// TIA Portal V16 export
// export: Created 2024-12-03T15:41:43.4866844Z, ExportSetting WithDefaults, DisplayName Totally Integrated Automation Portal, DisplayVersion V16 Update 6, DisplayName TIA Portal Version Control Interface, DisplayVersion V16 Update 2, DisplayName TIA Portal Openness, DisplayVersion V16 Update 6, DisplayName TIA Portal Teamcenter Gateway, DisplayVersion V16, DisplayName SINAMICS Startdrive Advanced, DisplayVersion V16 Update 5, DisplayName SINAMICS Startdrive G130, G150, S120, S150, SINAMICS MV, S210, DisplayVersion V16 Update 5, DisplayName SINAMICS Startdrive G110M, G120, G120C, G120D, G120P, G115D, DisplayVersion V16 Update 5, DisplayName STEP 7 Professional, DisplayVersion V16 Update 6, DisplayName STEP 7 Safety, DisplayVersion V16, DisplayName WinCC Advanced / Unified PC, DisplayVersion V16 Update 6
FUNCTION_BLOCK "IPC_Request"   // FB111, SCL
{ S7_Optimized_Access := 'TRUE' }
VERSION : 0.1
// stored: AutoNumber true, IsIECCheckEnabled false, IsRetainMemResEnabled false, MemoryReserve 100, SetENOAutomatically false, UDAEnableTagReadback false
   VAR_INPUT
      I_StartRequestFlag : Bool;
      I_AbortResend : Bool;
      I_Data : Variant;
      I_ResStatus { ExternalAccessible := 'False'; ExternalVisible := 'False'; ExternalWritable := 'False'} : "PLC_IPC_STANDARD_REQ_RES_UDT";
      I_ResData : Variant;
   END_VAR
   VAR_IN_OUT
      IO_IPC_Interface : "IPC_INTERFACE_STATUS_UDT";
      IO_ReqStatus : "PLC_IPC_STANDARD_REQ_RES_UDT";
      IO_ReqData : Variant;
      IO_ResultData : Variant;
   END_VAR
   VAR
      Alarm : "AlarmInfo_UDT";
      TriggerReader : "SmartBool";
      StepNumber : DInt := 100;
      MessageID : UInt := 1;
      Step_100_SentData : "StepperController";
      Step_200_ReceiveData : "StepperController";
      Step_300_ResendingPhase { S7_SetPoint := 'True'} : "StepperController";
      wmsError { S7_SetPoint := 'True'} : TON_TIME;
      alarmWmsError { S7_SetPoint := 'True'} : Program_Alarm;
   END_VAR
   VAR_TEMP
      T_ZoneInfo : "ZoneInfo";
      T_Condition : Bool;
      T_ErrorCondition : Bool;
      T_Res : Int;
   END_VAR
BEGIN
   REGION INIT
       #T_ZoneInfo := "ApplicationState_DB".ZoneNames[#IO_IPC_Interface.Zone];
   END_REGION

   REGION clear flags
       #IO_IPC_Interface.ResultStatus.pulse.Fail := 0;
       #IO_IPC_Interface.ResultStatus.pulse.Success := 0;
       #IO_IPC_Interface.ResultStatus.pulse.NewResult := 0;
       #IO_IPC_Interface.ResultStatus.pulse.TimeOut := 0;
       #IO_IPC_Interface.ResultStatus.pulse.OutOfSync := 0;
   END_REGION

   REGION Read trigger

       #TriggerReader(I_Sensor := #I_StartRequestFlag);

   END_REGION

   REGION Init step
       IF #StepNumber < 100 OR #StepNumber > 300 THEN
           #StepNumber := 100;
       END_IF;

   END_REGION

   REGION limit messageID
       IF #MessageID > 99999 THEN
           #MessageID := 1;
       END_IF;
   END_REGION

   REGION Init receive data flag when in step 100

       IF #StepNumber = 100 THEN
           //#IO_ResStatus.newData := 0;
           //#IO_ResStatus.messageId := 0;
           #IO_IPC_Interface.Settings.RetryCounter := 0;


           #IO_ReqStatus.newData := 0;

           RESET_TIMER(#Step_200_ReceiveData.S_TimeOutTime);
       END_IF;

   END_REGION

   REGION Step 100 standby waiting for sending trigger

       #Step_100_SentData(I_StepNumber := 100,
                          I_NextStepNumber := 200,
                          I_Condition := #TriggerReader.O_data.LE AND NOT #I_ResStatus.newData,
                          I_IgnoreTimeOut := TRUE,
                          IO_StepNumber := #StepNumber);

       IF #Step_100_SentData.O_ConditionTrans OR #Step_100_SentData.O_ErrorTrans THEN

           #T_Res := MOVE_BLK_VARIANT(SRC := #I_Data, COUNT := 1, SRC_INDEX := 0, DEST_INDEX := 0, DEST => #IO_ReqData);

           #IO_ReqStatus.messageId := #MessageID;
           #IO_ReqStatus.newData := TRUE;

           //Update message ID for next cycle
           #MessageID := #MessageID + 1;

       END_IF;

   END_REGION

   REGION Step 200 wait FOR receiving data

       #T_Condition := #I_ResStatus.newData
       AND #IO_ReqStatus.messageId = #I_ResStatus.messageId;

       #T_ErrorCondition := #I_ResStatus.newData
       AND #IO_ReqStatus.messageId <> #I_ResStatus.messageId;

       #Step_200_ReceiveData(I_StepNumber := 200,
                           I_NextStepNumber := 100,
                           I_TimeOutStepNumber:=300,
                           I_ErrorStepNumber := 300,
                           I_ErrorConditon := #T_ErrorCondition,
                           I_ErrorTime:= t#100ms,
                           I_ConditionTIme := t#100ms,
                           I_Condition := #T_Condition ,
                           I_TimeOutTime:=#IO_IPC_Interface.Settings.TimeOut,
                           I_IgnoreTimeOut := FALSE,
                           IO_StepNumber := #StepNumber);

   IF #StepNumber = 200 THEN
       //Log communication time
       #IO_IPC_Interface.Diagnostics.CommunicationTime := #Step_200_ReceiveData.S_TimeOutTime.ET;
   END_IF;




   END_REGION

   REGION TRANSITIONS

       REGION Succes transitions

           IF #Step_200_ReceiveData.O_ConditionTrans THEN

               //Update with new received data
               #T_Res := MOVE_BLK_VARIANT(SRC := #I_ResData, COUNT := 1, SRC_INDEX := 0, DEST_INDEX := 0, DEST => #IO_ResultData);

               //Acknowledge new data
               //#IO_ResStatus.newData := 0;

               //Update status bools
               #IO_IPC_Interface.ResultStatus.pulse.Success := TRUE;

               //Update diagnostics
               #IO_IPC_Interface.Diagnostics.Successes := #IO_IPC_Interface.Diagnostics.Successes + 1;

           END_IF;

       END_REGION

       REGION Failed transition

           IF #Step_200_ReceiveData.O_ErrorTrans OR #Step_200_ReceiveData.O_TimeTrans THEN

               //Acknowledge new data
               //#IO_ResStatus.newData := FALSE;

               //Update diagnostics
               IF #Step_200_ReceiveData.O_ErrorTrans THEN
                   #IO_IPC_Interface.Diagnostics.OutOfSync := #IO_IPC_Interface.Diagnostics.OutOfSync + 1;
               END_IF;

               IF #Step_200_ReceiveData.O_TimeTrans THEN
                   #IO_IPC_Interface.Diagnostics.TimeOuts := #IO_IPC_Interface.Diagnostics.TimeOuts + 1;
               END_IF;

           END_IF;

       END_REGION

       IF #Step_200_ReceiveData.O_ConditionTrans OR #Step_200_ReceiveData.O_ErrorTrans OR #Step_200_ReceiveData.O_TimeTrans THEN
           #IO_ReqStatus.newData := 0;
           #IO_ReqStatus.messageId := 0;
       END_IF;

   END_REGION

   REGION STEP 300 RESENT OBJECT

       #T_Condition := #IO_IPC_Interface.Settings.RetryCounter <= #IO_IPC_Interface.Settings.RetryThreshold
       AND #IO_IPC_Interface.Settings.RetrySending;

       #T_ErrorCondition := NOT #IO_IPC_Interface.Settings.RetrySending OR
       #I_AbortResend OR
       #IO_IPC_Interface.Settings.RetryCounter > #IO_IPC_Interface.Settings.RetryThreshold;

       #Step_300_ResendingPhase(I_StepNumber:=300,
                                I_NextStepNumber:=200,
                                I_ErrorStepNumber:=100,
                                I_TimeOutStepNumber:=100,
                                I_ErrorConditon := #T_ErrorCondition,
                                I_ErrorTime := t#0ms,
                                I_ConditionTIme := #IO_IPC_Interface.Settings.ResendMessage,
                                I_Condition:=#T_Condition,
                                I_IgnoreTimeOut:=TRUE,
                                IO_StepNumber:=#StepNumber);

       REGION RESENT PHASE

           IF #Step_300_ResendingPhase.O_ConditionTrans THEN

               //Retrigger message with current data
               #IO_ReqStatus.messageId := #MessageID;
               #IO_ReqStatus.newData := TRUE;

               //Update message ID for next cycle
               #MessageID := #MessageID + 1;

               #IO_IPC_Interface.Settings.RetryCounter += 1;

           END_IF;

       END_REGION

       REGION FAILED / RETRY THRESHOLD

           IF #Step_300_ResendingPhase.O_ErrorTrans THEN

               IF #Step_200_ReceiveData.O_ErrorTrans THEN
                   #IO_IPC_Interface.ResultStatus.pulse.OutOfSync := 1;
               END_IF;

               IF #Step_200_ReceiveData.O_TimeTrans THEN
                   #IO_IPC_Interface.ResultStatus.pulse.TimeOut := 1;
               END_IF;

               #IO_IPC_Interface.ResultStatus.pulse.Fail := 1;

           END_IF;

       END_REGION

   END_REGION

   REGION Update results statics

       IF #Step_200_ReceiveData.O_ConditionTrans
           OR (#Step_300_ResendingPhase.O_ErrorTrans
           AND (#Step_200_ReceiveData.O_ErrorTrans OR #Step_200_ReceiveData.O_TimeTrans)) THEN

           #IO_IPC_Interface.ResultStatus.pulse.NewResult := TRUE;
           #IO_IPC_Interface.ResultStatus.static := #IO_IPC_Interface.ResultStatus.pulse;
           #IO_IPC_Interface.Diagnostics.LastCommunicationTime := #IO_IPC_Interface.Diagnostics.CommunicationTime;

       END_IF;

   END_REGION

   REGION Update status

       #IO_IPC_Interface.Status.ReadyForSendingData := #StepNumber = 100 AND NOT #I_ResStatus.newData;
       #IO_IPC_Interface.Status.ReceivingData := #StepNumber = 200 OR #StepNumber = 300;

   END_REGION

   REGION ALARAM

       REGION INFO

           //#IO_IPC_Interface.name := "buildObjectName"(I_Symbolname := GetSymbolName(variable := #IO_IPC_Interface, size := 200));

           IF NOT #Alarm.init OR #IO_IPC_Interface.name = '' OR #Alarm.info = '' OR "HMI_DB".ReloadSettings.signal THEN
               //#IO_IPC_Interface.name := "buildObjectName"(I_Symbolname := GetSymbolName(variable := #IO_IPC_Interface, size := 200));
                   #Alarm.info := "buildAlarmInfo"(I_ObjectName := #IO_IPC_Interface.name, I_ZoneIndex := #IO_IPC_Interface.Zone, I_ZoneName := #T_ZoneInfo.ZoneName);
                   #Alarm.init := true;
               END_IF;
       END_REGION

       //Trigger alarm when new data are active for to long
       #wmsError(IN:= NOT #IO_ReqStatus.newData AND #I_ResStatus.newData,
                 PT:=t#10s);

       #alarmWmsError(SIG:=#wmsError.Q, SD_1 := #IO_IPC_Interface.name, SD_2 := #Alarm.info);

   END_REGION

   REGION SETTINGS

       #IO_IPC_Interface.Settings.TimeOut := t#15s;
       #IO_IPC_Interface.Settings.RetrySending := 1;
       #IO_IPC_Interface.Settings.RetryThreshold := 5;
       #IO_IPC_Interface.Settings.ResendMessage := T#3S;

   END_REGION
END_FUNCTION_BLOCK
